// TwinCAT 3 PLC project demo
// libraries:
//   Tc2_Standard, * (Beckhoff Automation GmbH)
//   Tc2_System, * (Beckhoff Automation GmbH)
//   Tc3_Interfaces, * (Beckhoff Automation GmbH)
//   Tc3_Module, * (Beckhoff Automation GmbH)
// project tree:
//   Data types/ ST_ChartFields.TcDUT, ST_Test.TcDUT, ST_Test2.TcDUT, ST_Test3.TcDUT, ST_Test4.TcDUT
//   Global Variables/ Globale_Variablen.TcGVL, Variablen_Konfiguration.TcGVL
//   POUs/FB%27s/ FB_Ramp.TcPOU (not stored), FB_RunningLight.TcPOU (not stored), FB_ShiftArray.TcPOU (not stored), TogRS.TcPOU (not stored)
//   POUs/ MAIN.TcPOU
//   / Standard.TcTTO

CONFIGURATION demo
    RESOURCE PLC ON TwinCAT3
        TASK Standard(INTERVAL := T#10ms, PRIORITY := 20);
        PROGRAM MAIN WITH Standard : MAIN;
    END_RESOURCE
END_CONFIGURATION

// ---- Data types/ST_ChartFields.TcDUT
TYPE ST_ChartFields :
STRUCT
	graph1: INT;
	graph2: INT;
END_STRUCT
END_TYPE

// ---- Data types/ST_Test.TcDUT
TYPE ST_Test :
STRUCT
	nByte: BYTE;
	fReal: REAL;
	iSint: SINT;
	tTime: TIME;
	arrString: ARRAY[1..5] OF STRING(6);
	iInt: INT;
END_STRUCT
END_TYPE

// ---- Data types/ST_Test2.TcDUT
TYPE ST_Test2 :
STRUCT
	sString: STRING(5) := 'xxxxx';
	fReal: REAL;
	iSint: SINT;
	iInt: INT;
	arrByte: ARRAY[1..5] OF BYTE;
END_STRUCT
END_TYPE

// ---- Data types/ST_Test3.TcDUT
TYPE ST_Test3 :
STRUCT
	sString: STRING(10) := '';
	fReal: REAL;
	iInt: INT;
	nByte: BYTE;
	bCheckbox: BOOL;
	arrBool: ARRAY[1..5] OF BOOL;
END_STRUCT
END_TYPE

// ---- Data types/ST_Test4.TcDUT
TYPE ST_Test4 :
STRUCT
	fReal: REAL;
	tTime: TIME;
	tTod: TOD;
	dtDate: DATE;
	arrString: ARRAY[1..5] OF STRING(6);
END_STRUCT
END_TYPE

// ---- Global Variables/Globale_Variablen.TcGVL
{attribute 'Tc2GvlVarNames'}
VAR_GLOBAL
	
	OUT_BOOL_1 AT %Q*:BOOL;
	OUT_BOOL_2 AT %Q*:BOOL;
	OUT_BOOL_3 AT %Q*:BOOL;
	OUT_BOOL_4 AT %Q*:BOOL;
	OUT_BOOL_5 AT %Q*:BOOL;
	OUT_BOOL_6 AT %Q*:BOOL;
	OUT_BOOL_7 AT %Q*:BOOL;
	OUT_BOOL_8 AT %Q*:BOOL;
	
	IN_BOOL_1 AT %I*:BOOL;
	IN_BOOL_2 AT %I*:BOOL;
	IN_BOOL_3 AT %I*:BOOL;
	IN_BOOL_4 AT %I*:BOOL;
	IN_BOOL_5 AT %I*:BOOL;
	IN_BOOL_6 AT %I*:BOOL;
	IN_BOOL_7 AT %I*:BOOL;
	IN_BOOL_8 AT %I*:BOOL;
	
	OUT_INT_1 AT %Q*:INT;
	OUT_INT_2 AT %Q*:INT;
	
	IN_INT_1 AT %I*:INT;
	IN_INT_2 AT %I*:INT;
	
	In_BOOL1 AT%MX0.0 : BOOL;
	In_BOOL2: BOOL;

	In_SINT1: SINT;
	In_SINT2: SINT;
	In_SINT3: SINT;
	In_SINT4: SINT;
	In_INT1: INT;
	In_INT2: INT;
	In_DINT: DINT;
	In_STRING: STRING(11);
	In_TIME: TIME;
	In_REAL: REAL;
	

	TOD_Test : TOD;
	DT_Test: DT;
	DATE_Test: DATE;

	ArrayOfString: ARRAY[1..5] OF STRING(10);
	ArrayOfBool:  ARRAY[1..5] OF BOOL;

	ArrayOfTestStruct2: ARRAY[1..4] OF ST_Test2;

	TestStruct:  ST_Test;

	ArrayTestStruct3: ARRAY [1..20] OF ST_Test3;

	TestStruct4 :  ST_Test4;

	ArrayChart: ARRAY [1..10] OF ST_ChartFields (*Kommentar*);
END_VAR

// ---- Global Variables/Variablen_Konfiguration.TcGVL
{attribute 'Tc2GvlVarNames'}
VAR_CONFIG
END_VAR

// ---- POUs/MAIN.TcPOU
PROGRAM MAIN
VAR
	fbRamp1: FB_Ramp;
	fbRamp2: FB_Ramp;
	fbShiftArray: FB_ShiftArray;
	fbRunningLight: FB_RunningLight;
	Ramp1 : INT;
	Ramp2 : INT;
	RunningLight1: BOOL;
	RunningLight2: BOOL;
	RunningLight3: BOOL;
	RunningLight4: BOOL;
	RunningLight5: BOOL;
	
END_VAR

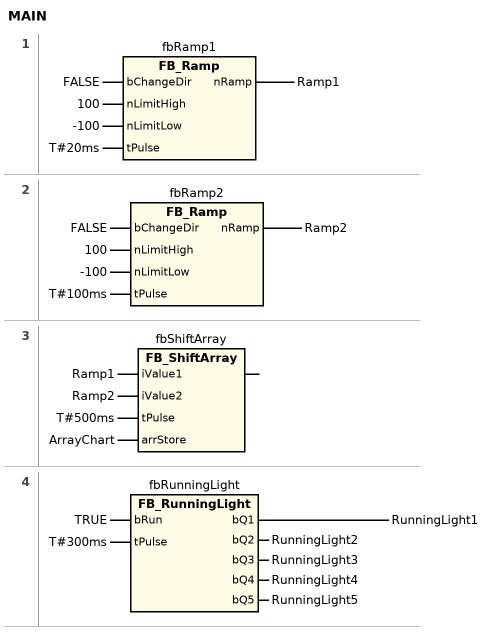
// NETWORK 1
fbRamp1(bChangeDir := FALSE, nLimitHigh := 100, nLimitLow := -100, tPulse := T#20ms); // FB_Ramp
Ramp1 := fbRamp1.nRamp;

// NETWORK 2
fbRamp2(bChangeDir := FALSE, nLimitHigh := 100, nLimitLow := -100, tPulse := T#100ms); // FB_Ramp
Ramp2 := fbRamp2.nRamp;

// NETWORK 3
fbShiftArray(iValue1 := Ramp1, iValue2 := Ramp2, tPulse := T#500ms, arrStore := ArrayChart); // FB_ShiftArray

// NETWORK 4
fbRunningLight(
    bRun := TRUE,
    tPulse := T#300ms,
    bQ2 => RunningLight2,
    bQ3 => RunningLight3,
    bQ4 => RunningLight4,
    bQ5 => RunningLight5); // FB_RunningLight
RunningLight1 := fbRunningLight.bQ1;

END_PROGRAM
